// TIA Portal V18 export
FUNCTION_BLOCK "artLimFormer"   // FB74, FBD
{ S7_Optimized_Access := 'TRUE' }
VERSION : 0.1
// stored: AutoNumber true, IsIECCheckEnabled false, IsRetainMemResEnabled false, MemoryReserve 100, SetENOAutomatically false, UDAEnableTagReadback false
   VAR_INPUT
      doors_open_fully : Bool;
      pos_x : Real;
      pos_y : Real;
      lim_yrev_chamber_doorsClosed_safe : Real;
      lim_x_fwd_outside : Real;
      lim_x_rev_outside : Real;
      normal_x_rev : Real;
      normal_x_fwd : Real;
      normal_y_rev : Real;
      normal_y_fwd : Real;
      margin_x : Real;
      ACK : Bool;
      margin_y : Real;
   END_VAR
   VAR_OUTPUT
      result_x_rev : Real;
      result_x_fwd : Real;
      result_y_rev : Real;
      result_y_fwd : Real;
      ER_WS : WString;
      ER : Bool;
      y_is_inside_safely : Bool;
   END_VAR
   VAR
      y_can_go_out_rev : Bool;
      x_fits_in_doors : Bool;
      y_is_inside : Bool;
   END_VAR
   VAR_TEMP
      lim_x_fwd_outside_p_margin : Real;
      loc_lim_x_fwd_outside_p_margin : Real;
      loc_lim_x_rev_outside_m_margin : Real;
      loc_lim_yrev_chamber_doorsClosed_safe_m_margin : Real;
   END_VAR
   VAR CONSTANT
      erws1 : WString := WSTRING#'wrong limits';
   END_VAR
BEGIN

REGION Network 1 (SCL)
   #loc_lim_x_fwd_outside_p_margin := #lim_x_fwd_outside + #margin_x;
   #loc_lim_x_rev_outside_m_margin := #lim_x_rev_outside - #margin_x; 

   #loc_lim_yrev_chamber_doorsClosed_safe_m_margin := #lim_yrev_chamber_doorsClosed_safe - #margin_y;
END_REGION

REGION Network 2
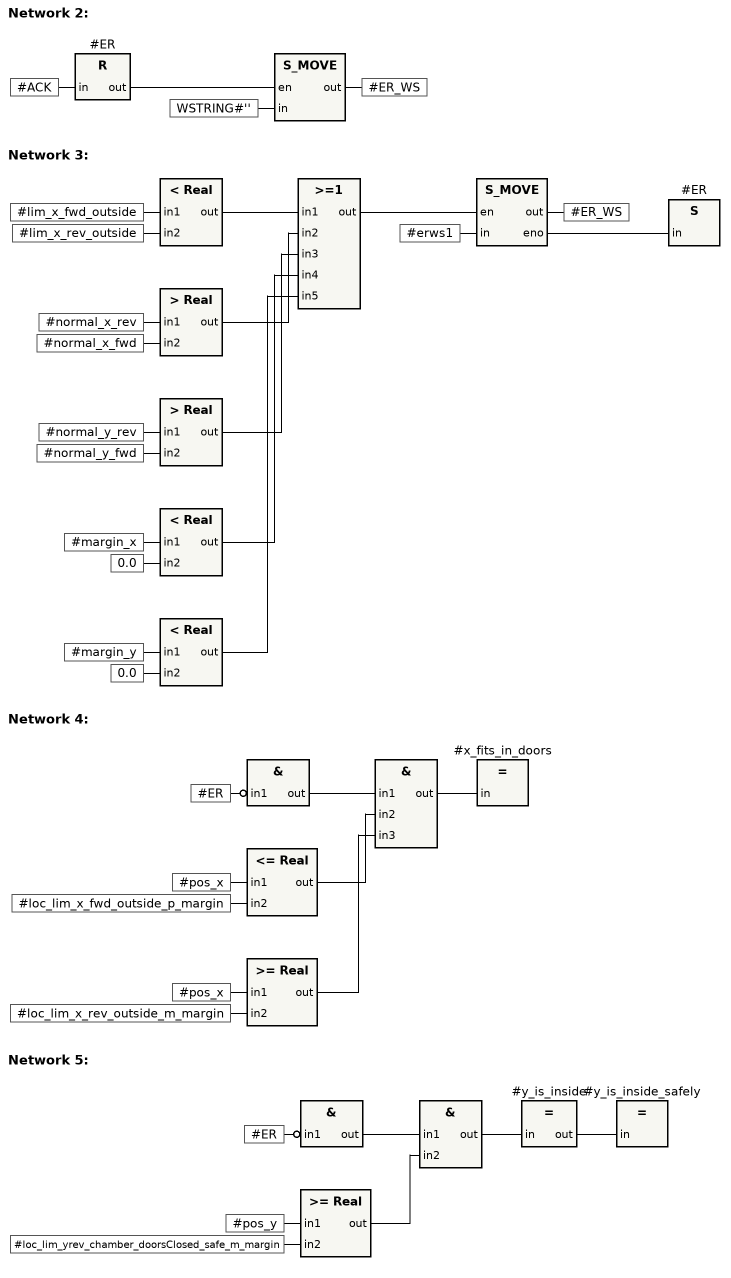
   IF #ACK THEN
       #ER := FALSE;
       #ER_WS := WSTRING#'';
   END_IF;
END_REGION

REGION Network 3
   IF (#lim_x_fwd_outside < #lim_x_rev_outside) OR (#normal_x_rev > #normal_x_fwd) OR (#normal_y_rev > #normal_y_fwd) OR (#margin_x < 0.0) OR (#margin_y < 0.0) THEN
       #ER_WS := #erws1;
       #ER := TRUE;
   END_IF;
END_REGION

REGION Network 4
   #x_fits_in_doors := NOT #ER AND (#pos_x <= #loc_lim_x_fwd_outside_p_margin) AND (#pos_x >= #loc_lim_x_rev_outside_m_margin);
END_REGION

REGION Network 5
   #y_is_inside := NOT #ER AND (#pos_y >= #loc_lim_yrev_chamber_doorsClosed_safe_m_margin);
   #y_is_inside_safely := #y_is_inside;
END_REGION

REGION Network 6
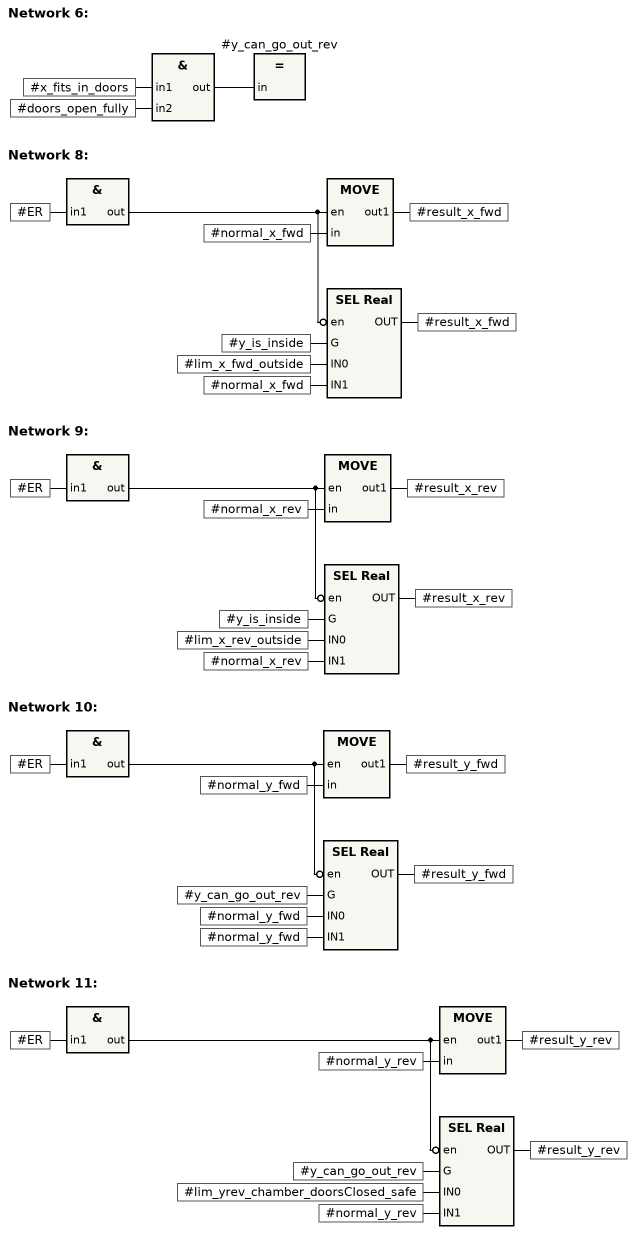
   #y_can_go_out_rev := #x_fits_in_doors AND #doors_open_fully;
END_REGION

REGION Network 8
   IF #ER THEN #result_x_fwd := #normal_x_fwd; END_IF;
   IF NOT #ER THEN
       #result_x_fwd := SEL(G := #y_is_inside, IN0 := #lim_x_fwd_outside, IN1 := #normal_x_fwd);
   END_IF;
END_REGION

REGION Network 9
   IF #ER THEN #result_x_rev := #normal_x_rev; END_IF;
   IF NOT #ER THEN
       #result_x_rev := SEL(G := #y_is_inside, IN0 := #lim_x_rev_outside, IN1 := #normal_x_rev);
   END_IF;
END_REGION

REGION Network 10
   IF #ER THEN #result_y_fwd := #normal_y_fwd; END_IF;
   IF NOT #ER THEN
       #result_y_fwd := SEL(G := #y_can_go_out_rev, IN0 := #normal_y_fwd, IN1 := #normal_y_fwd);
   END_IF;
END_REGION

REGION Network 11
   IF #ER THEN #result_y_rev := #normal_y_rev; END_IF;
   IF NOT #ER THEN
       #result_y_rev := SEL(G := #y_can_go_out_rev, IN0 := #lim_yrev_chamber_doorsClosed_safe, IN1 := #normal_y_rev);
   END_IF;
END_REGION
END_FUNCTION_BLOCK
